// TIA Portal project "HeThongSanXuatTraXanh" (V16)

(* hardware
DEVICE "S7-1200 station_1"  S7-1200 Station
   slot 0: "Rack_0"  S7-1200 Rack  Rack  V1.0
   slot 1: "PLC_1"  CPU 1212C AC/DC/Rly  6ES7 212-1BE40-0XB0  V4.4
DEVICE "PC-System_1"  SIMATIC PC station
   slot 0: "SIMATIC PC station"  Rail  SIMATIC PC-Station  V1.0
      slot 125: "Stationmanager"  Station_Manager  V6.0.4
   slot 1: "HMI_RT_1"  WinCC RT Advanced  6AV2 104-0xxxx-xxxx  16.0.0.0
      slot 33792: "Computer interface"  Host interface
   slot 2: "IE general_1"  IE General  IE_CP  V8.2.0
*)

// ===== PLC "PLC_1"  CPU 1212C AC/DC/Rly =====

VAR_GLOBAL   // PLC tag table "Default tag table"
   "System_Byte" AT %MB1 : Byte;
   "FirstScan" AT %M1.0 : Bool;
   "DiagStatusUpdate" AT %M1.1 : Bool;
   "AlwaysTRUE" AT %M1.2 : Bool;
   "AlwaysFALSE" AT %M1.3 : Bool;
   "Clock_Byte" AT %MB0 : Byte;
   "Clock_10Hz" AT %M0.0 : Bool;
   "Clock_5Hz" AT %M0.1 : Bool;
   "Clock_2.5Hz" AT %M0.2 : Bool;
   "Clock_2Hz" AT %M0.3 : Bool;
   "Clock_1.25Hz" AT %M0.4 : Bool;
   "Clock_1Hz" AT %M0.5 : Bool;
   "Clock_0.625Hz" AT %M0.6 : Bool;
   "Clock_0.5Hz" AT %M0.7 : Bool;
   "alarm_word" AT %MW20 : Word;
   "alarm1" AT %M20.0 : Bool;
   "alarm2" AT %M20.1 : Bool;
END_VAR

VAR_GLOBAL   // PLC tag table "INPUT"
   "I_Mode" AT %I0.0 : Bool;
   "I_Auto_Run" AT %I0.1 : Bool;
   "I_Auto_Stop" AT %I0.2 : Bool;
   "I_BT1" AT %I0.3 : Bool;
   "I_BT2" AT %I0.4 : Bool;
   "I_BT3" AT %I0.5 : Bool;
   "I_BT4" AT %I0.6 : Bool;
   "I_BT5" AT %I0.7 : Bool;
   "I_BT6" AT %I1.0 : Bool;
   "I_Valve1" AT %I1.1 : Bool;
   "I_May_Hap" AT %I1.2 : Bool;
   "I_May_Vo" AT %I1.3 : Bool;
   "I_May_Say" AT %I1.4 : Bool;
   "I_May_Sang" AT %I1.5 : Bool;
   "I_May_Dong_Goi" AT %I1.6 : Bool;
   "IW_Loadcell" AT %IW64 : Int;
   "IW_Temp_Hap" AT %IW66 : Int;
   "IW_Temp_Say" AT %IW68 : Int;
END_VAR

VAR_GLOBAL   // PLC tag table "OUTPUT"
   "Q_Lamp_Auto" AT %Q0.0 : Bool;
   "Q_Lamp_Manu" AT %Q0.1 : Bool;
   "Q_Lamp_Auto_Running" AT %Q0.2 : Bool;
   "Q_BT1" AT %Q0.3 : Bool;
   "Q_BT2" AT %Q0.4 : Bool;
   "Q_BT3" AT %Q0.5 : Bool;
   "Q_BT4" AT %Q0.6 : Bool;
   "Q_BT5" AT %Q0.7 : Bool;
   "Q_BT6" AT %Q1.0 : Bool;
   "Q_Valve1" AT %Q1.1 : Bool;
   "Q_May_Hap" AT %Q1.2 : Bool;
   "Q_May_Vo" AT %Q1.3 : Bool;
   "Q_May_Say" AT %Q1.4 : Bool;
   "Q_May_Sang" AT %Q1.5 : Bool;
   "Q_May_Dong_Goi" AT %Q1.6 : Bool;
END_VAR

VAR_GLOBAL   // PLC tag table "MIEN_NHO"
   "Set_Weight" AT %MD100 : Real;
   "Set_Temp_Hap" AT %MD104 : Real;
   "Set_Temp_Say" AT %MD108 : Real;
   "Act_Weight" AT %MD200 : Real;
   "Act_Temp_Hap" AT %MD204 : Real;
   "Act_Temp_Say" AT %MD208 : Real;
   "Act_San_Luong" AT %MW212 : Int;
   "Simu_Temp" AT %MD220 : Real;
END_VAR

VAR_GLOBAL   // PLC tag table "TRUNG_GIAN"
   "Q_Auto_BT1" AT %M20.0 : Bool;
   "Q_Auto_BT2" AT %M20.1 : Bool;
   "Q_Auto_BT3" AT %M20.2 : Bool;
   "Q_Auto_BT4" AT %M20.3 : Bool;
   "Q_Auto_BT5" AT %M20.4 : Bool;
   "Q_Auto_BT6" AT %M20.5 : Bool;
   "Q_Auto_Valve1" AT %M20.6 : Bool;
   "Q_Auto_May_Hap" AT %M20.7 : Bool;
   "Q_Auto_May_Vo" AT %M21.0 : Bool;
   "Q_Auto_May_Say" AT %M21.1 : Bool;
   "Q_Auto_May_Sang" AT %M21.2 : Bool;
   "Q_Auto_May_Dong_Goi" AT %M21.3 : Bool;
   "Q_Manu_BT1" AT %M30.0 : Bool;
   "Q_Manu_BT2" AT %M30.1 : Bool;
   "Q_Manu_BT3" AT %M30.2 : Bool;
   "Q_Manu_BT4" AT %M30.3 : Bool;
   "Q_Manu_BT5" AT %M30.4 : Bool;
   "Q_Manu_BT6" AT %M30.5 : Bool;
   "Q_Manu_Valve1" AT %M30.6 : Bool;
   "Q_Manu_May_Hap" AT %M30.7 : Bool;
   "Q_Manu_May_Vo" AT %M31.0 : Bool;
   "Q_Manu_May_Say" AT %M31.1 : Bool;
   "Q_Manu_May_Sang" AT %M31.2 : Bool;
   "Q_Manu_May_Dong_Goi" AT %M31.3 : Bool;
END_VAR

VAR_GLOBAL   // PLC tag table "M"
   "M_Mode" AT %M10.0 : Bool;
   "M_Auto_Run" AT %M10.1 : Bool;
   "M_Auto_Stop" AT %M10.2 : Bool;
   "M_BT1" AT %M10.3 : Bool;
   "M_BT2" AT %M10.4 : Bool;
   "M_BT3" AT %M10.5 : Bool;
   "M_BT4" AT %M10.6 : Bool;
   "M_BT5" AT %M10.7 : Bool;
   "M_BT6" AT %M11.0 : Bool;
   "M_Valve1" AT %M11.1 : Bool;
   "M_May_Hap" AT %M11.2 : Bool;
   "M_May_Vo" AT %M11.3 : Bool;
   "M_May_Say" AT %M11.4 : Bool;
   "M_May_Sang" AT %M11.5 : Bool;
   "M_May_Dong_Goi" AT %M11.6 : Bool;
   "MW_Loadcell" AT %MW64 : Int;
   "MW_Temp_Hap" AT %MW66 : Int;
   "MW_Temp_Say" AT %MW68 : Int;
   "M_Simulation" AT %M5.0 : Bool;
END_VAR

VAR_GLOBAL   // PLC tag table "STEP"
   "STEP_1" AT %M40.0 : Bool;
   "STEP_2" AT %M40.1 : Bool;
   "STEP_3" AT %M40.2 : Bool;
   "STEP_4" AT %M40.3 : Bool;
   "STEP_5" AT %M40.4 : Bool;
   "STEP_6" AT %M40.5 : Bool;
   "STEP_7" AT %M40.6 : Bool;
   "STEP_8" AT %M40.7 : Bool;
   "STEP_9" AT %M41.0 : Bool;
   "STEP_10" AT %M41.1 : Bool;
   "STEP_11" AT %M41.2 : Bool;
END_VAR

VAR_GLOBAL   // PLC tag table "XUNG P"
   "P1" AT %M90.0 : Bool;
   "P2" AT %M90.1 : Bool;
   "P3" AT %M90.2 : Bool;
   "P4" AT %M90.3 : Bool;
   "P5" AT %M90.4 : Bool;
   "P6" AT %M90.5 : Bool;
   "P7" AT %M90.6 : Bool;
   "P8" AT %M90.7 : Bool;
   "P9" AT %M91.0 : Bool;
   "P10" AT %M91.1 : Bool;
   "P11" AT %M91.2 : Bool;
   "P12" AT %M91.3 : Bool;
   "P13" AT %M91.4 : Bool;
   "P14" AT %M91.5 : Bool;
   "P15" AT %M91.6 : Bool;
   "P16" AT %M91.7 : Bool;
   "P17" AT %M92.0 : Bool;
   "P18" AT %M92.1 : Bool;
   "P19" AT %M92.2 : Bool;
   "P20" AT %M92.3 : Bool;
END_VAR

// folder: System blocks/Program resources

DATA_BLOCK "TIMER_STEP2"   // DB1
{ S7_Optimized_Access := 'TRUE' }
AUTHOR : Simatic
FAMILY : IEC
NAME : IEC_TMR
VERSION : 1.0
// stored: InstanceOfName IEC_TIMER
"IEC_TIMER"
BEGIN
END_DATA_BLOCK

DATA_BLOCK "TIMER_STEP3"   // DB2
{ S7_Optimized_Access := 'TRUE' }
AUTHOR : Simatic
FAMILY : IEC
NAME : IEC_TMR
VERSION : 1.0
// stored: InstanceOfName IEC_TIMER
"IEC_TIMER"
BEGIN
END_DATA_BLOCK

DATA_BLOCK "TIMER_STEP4"   // DB3
{ S7_Optimized_Access := 'TRUE' }
AUTHOR : Simatic
FAMILY : IEC
NAME : IEC_TMR
VERSION : 1.0
// stored: InstanceOfName IEC_TIMER
"IEC_TIMER"
BEGIN
END_DATA_BLOCK

DATA_BLOCK "TIMER_STEP5"   // DB4
{ S7_Optimized_Access := 'TRUE' }
AUTHOR : Simatic
FAMILY : IEC
NAME : IEC_TMR
VERSION : 1.0
// stored: InstanceOfName IEC_TIMER
"IEC_TIMER"
BEGIN
END_DATA_BLOCK

DATA_BLOCK "TIMER_STEP6"   // DB5
{ S7_Optimized_Access := 'TRUE' }
AUTHOR : Simatic
FAMILY : IEC
NAME : IEC_TMR
VERSION : 1.0
// stored: InstanceOfName IEC_TIMER
"IEC_TIMER"
BEGIN
END_DATA_BLOCK

DATA_BLOCK "TIMER_STEP7"   // DB6
{ S7_Optimized_Access := 'TRUE' }
AUTHOR : Simatic
FAMILY : IEC
NAME : IEC_TMR
VERSION : 1.0
// stored: InstanceOfName IEC_TIMER
"IEC_TIMER"
BEGIN
END_DATA_BLOCK

DATA_BLOCK "TIMER_STEP8"   // DB7
{ S7_Optimized_Access := 'TRUE' }
AUTHOR : Simatic
FAMILY : IEC
NAME : IEC_TMR
VERSION : 1.0
// stored: InstanceOfName IEC_TIMER
"IEC_TIMER"
BEGIN
END_DATA_BLOCK

DATA_BLOCK "TIMER_STEP9"   // DB8
{ S7_Optimized_Access := 'TRUE' }
AUTHOR : Simatic
FAMILY : IEC
NAME : IEC_TMR
VERSION : 1.0
// stored: InstanceOfName IEC_TIMER
"IEC_TIMER"
BEGIN
END_DATA_BLOCK

DATA_BLOCK "TIMER_STEP10"   // DB9
{ S7_Optimized_Access := 'TRUE' }
AUTHOR : Simatic
FAMILY : IEC
NAME : IEC_TMR
VERSION : 1.0
// stored: InstanceOfName IEC_TIMER
"IEC_TIMER"
BEGIN
END_DATA_BLOCK

DATA_BLOCK "TIMER_STEP11"   // DB10
{ S7_Optimized_Access := 'TRUE' }
AUTHOR : Simatic
FAMILY : IEC
NAME : IEC_TMR
VERSION : 1.0
// stored: InstanceOfName IEC_TIMER
"IEC_TIMER"
BEGIN
END_DATA_BLOCK

// folder: (top level)

FUNCTION "FC_AUTO_MODE" : Void   // FC1, LAD
{ S7_Optimized_Access := 'TRUE' }
VERSION : 0.1
   VAR_TEMP   // added for the SCL form of the ladder/FBD networks
      _w1 : Bool;
      _w2 : Bool;
   END_VAR
BEGIN

REGION Network 1
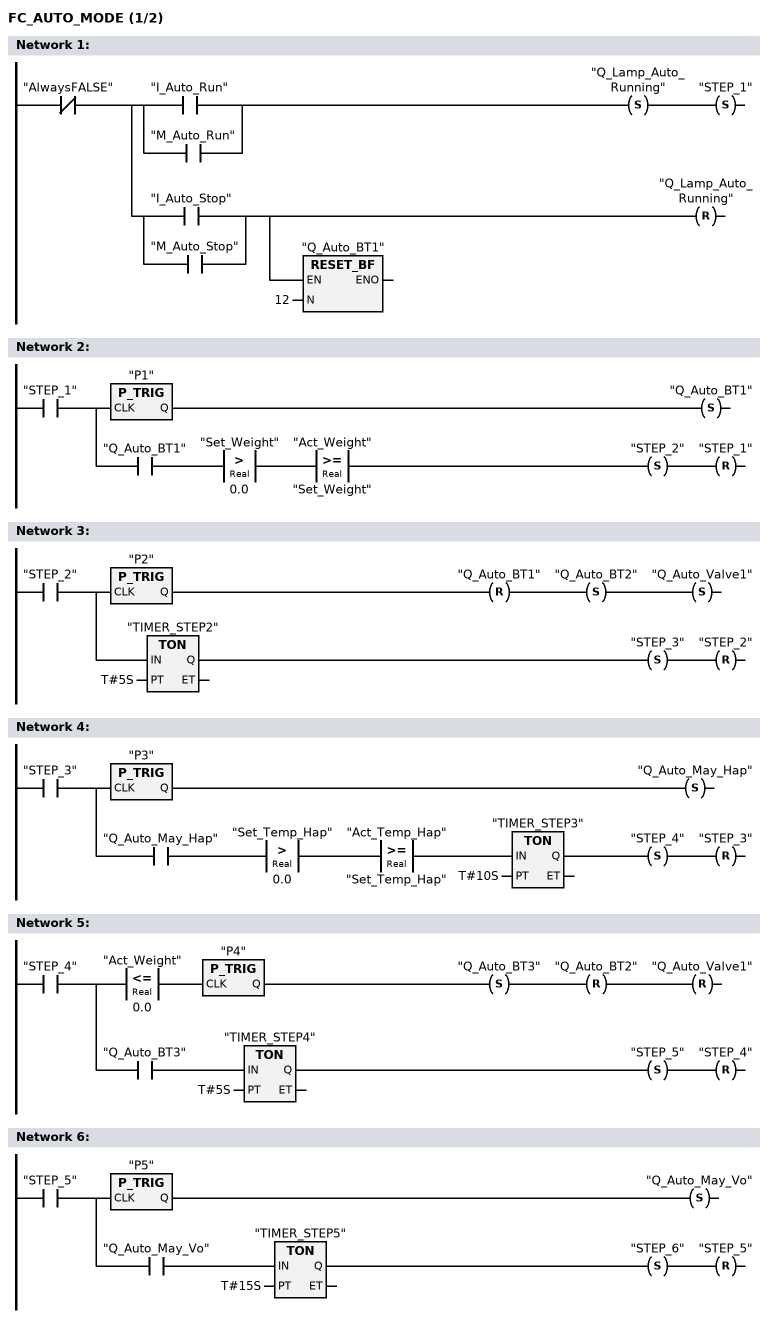
   // no SCL statement known for RBitfield: written as a call
   IF NOT "AlwaysFALSE" AND ("I_Auto_Run" OR "M_Auto_Run") THEN
       "Q_Lamp_Auto_Running" := TRUE;
       "STEP_1" := TRUE;
   END_IF;
   IF NOT "AlwaysFALSE" AND ("I_Auto_Stop" OR "M_Auto_Stop") THEN
       "Q_Lamp_Auto_Running" := FALSE;
       RESET_BF(operand := "Q_Auto_BT1", n := 12);
   END_IF;
END_REGION

REGION Network 2
   RUNG wire#powerrail
      Contact( "STEP_1" )
      wire#w1
      P_Trig( "P1" )
      S_Coil( "Q_Auto_BT1" )
   END_RUNG
   RUNG wire#w1
      Contact( "Q_Auto_BT1" )
      { S7_Templates := "SrcType := Real" } GT_Contact(in1 := "Set_Weight", in2 := 0.0)
      { S7_Templates := "SrcType := Real" } GE_Contact(in1 := "Act_Weight", in2 := "Set_Weight")
      S_Coil( "STEP_2" )
      R_Coil( "STEP_1" )
   END_RUNG
   // the same network as SCL:
   #_w1 := "STEP_1" AND NOT "P1";   // rising edge
   "P1" := "STEP_1";
   IF #_w1 THEN "Q_Auto_BT1" := TRUE; END_IF;
   IF "STEP_1" AND "Q_Auto_BT1" AND ("Set_Weight" > 0.0) AND ("Act_Weight" >= "Set_Weight") THEN
       "STEP_2" := TRUE;
       "STEP_1" := FALSE;
   END_IF;
END_REGION

REGION Network 3
   #_w1 := "STEP_2" AND NOT "P2";   // rising edge
   "P2" := "STEP_2";
   IF #_w1 THEN
       "Q_Auto_BT1" := FALSE;
       "Q_Auto_BT2" := TRUE;
       "Q_Auto_Valve1" := TRUE;
   END_IF;
   "TIMER_STEP2".TON(IN := "STEP_2", PT := T#5S);
   IF "TIMER_STEP2".Q THEN
       "STEP_3" := TRUE;
       "STEP_2" := FALSE;
   END_IF;
END_REGION

REGION Network 4
   #_w1 := "STEP_3" AND NOT "P3";   // rising edge
   "P3" := "STEP_3";
   IF #_w1 THEN "Q_Auto_May_Hap" := TRUE; END_IF;
   "TIMER_STEP3".TON(IN := "STEP_3" AND "Q_Auto_May_Hap" AND ("Set_Temp_Hap" > 0.0) AND ("Act_Temp_Hap" >= "Set_Temp_Hap"),
                     PT := T#10S);
   IF "TIMER_STEP3".Q THEN
       "STEP_4" := TRUE;
       "STEP_3" := FALSE;
   END_IF;
END_REGION

REGION Network 5
   #_w1 := "STEP_4" AND ("Act_Weight" <= 0.0);
   #_w2 := #_w1 AND NOT "P4";   // rising edge
   "P4" := #_w1;
   IF #_w2 THEN
       "Q_Auto_BT3" := TRUE;
       "Q_Auto_BT2" := FALSE;
       "Q_Auto_Valve1" := FALSE;
   END_IF;
   "TIMER_STEP4".TON(IN := "STEP_4" AND "Q_Auto_BT3", PT := T#5S);
   IF "TIMER_STEP4".Q THEN
       "STEP_5" := TRUE;
       "STEP_4" := FALSE;
   END_IF;
END_REGION

REGION Network 6
   #_w1 := "STEP_5" AND NOT "P5";   // rising edge
   "P5" := "STEP_5";
   IF #_w1 THEN "Q_Auto_May_Vo" := TRUE; END_IF;
   "TIMER_STEP5".TON(IN := "STEP_5" AND "Q_Auto_May_Vo", PT := T#15S);
   IF "TIMER_STEP5".Q THEN
       "STEP_6" := TRUE;
       "STEP_5" := FALSE;
   END_IF;
END_REGION

REGION Network 7
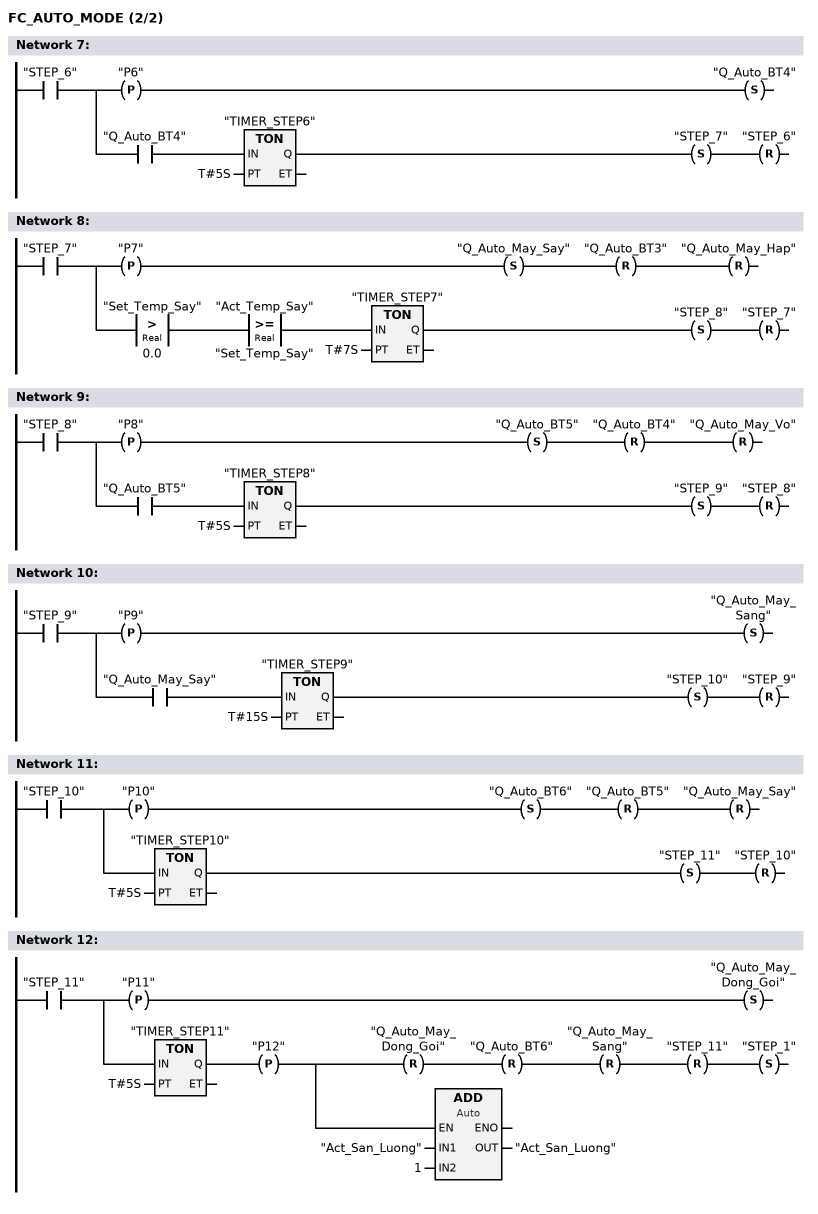
   #_w1 := "STEP_6" AND NOT "P6";   // rising edge
   "P6" := "STEP_6";
   IF #_w1 THEN "Q_Auto_BT4" := TRUE; END_IF;
   "TIMER_STEP6".TON(IN := "STEP_6" AND "Q_Auto_BT4", PT := T#5S);
   IF "TIMER_STEP6".Q THEN
       "STEP_7" := TRUE;
       "STEP_6" := FALSE;
   END_IF;
END_REGION

REGION Network 8
   #_w1 := "STEP_7" AND NOT "P7";   // rising edge
   "P7" := "STEP_7";
   IF #_w1 THEN
       "Q_Auto_May_Say" := TRUE;
       "Q_Auto_BT3" := FALSE;
       "Q_Auto_May_Hap" := FALSE;
   END_IF;
   "TIMER_STEP7".TON(IN := "STEP_7" AND ("Set_Temp_Say" > 0.0) AND ("Act_Temp_Say" >= "Set_Temp_Say"),
                     PT := T#7S);
   IF "TIMER_STEP7".Q THEN
       "STEP_8" := TRUE;
       "STEP_7" := FALSE;
   END_IF;
END_REGION

REGION Network 9
   #_w1 := "STEP_8" AND NOT "P8";   // rising edge
   "P8" := "STEP_8";
   IF #_w1 THEN
       "Q_Auto_BT5" := TRUE;
       "Q_Auto_BT4" := FALSE;
       "Q_Auto_May_Vo" := FALSE;
   END_IF;
   "TIMER_STEP8".TON(IN := "STEP_8" AND "Q_Auto_BT5", PT := T#5S);
   IF "TIMER_STEP8".Q THEN
       "STEP_9" := TRUE;
       "STEP_8" := FALSE;
   END_IF;
END_REGION

REGION Network 10
   #_w1 := "STEP_9" AND NOT "P9";   // rising edge
   "P9" := "STEP_9";
   IF #_w1 THEN "Q_Auto_May_Sang" := TRUE; END_IF;
   "TIMER_STEP9".TON(IN := "STEP_9" AND "Q_Auto_May_Say", PT := T#15S);
   IF "TIMER_STEP9".Q THEN
       "STEP_10" := TRUE;
       "STEP_9" := FALSE;
   END_IF;
END_REGION

REGION Network 11
   #_w1 := "STEP_10" AND NOT "P10";   // rising edge
   "P10" := "STEP_10";
   IF #_w1 THEN
       "Q_Auto_BT6" := TRUE;
       "Q_Auto_BT5" := FALSE;
       "Q_Auto_May_Say" := FALSE;
   END_IF;
   "TIMER_STEP10".TON(IN := "STEP_10", PT := T#5S);
   IF "TIMER_STEP10".Q THEN
       "STEP_11" := TRUE;
       "STEP_10" := FALSE;
   END_IF;
END_REGION

REGION Network 12
   #_w1 := "STEP_11" AND NOT "P11";   // rising edge
   "P11" := "STEP_11";
   IF #_w1 THEN "Q_Auto_May_Dong_Goi" := TRUE; END_IF;
   "TIMER_STEP11".TON(IN := "STEP_11", PT := T#5S);
   #_w2 := "TIMER_STEP11".Q AND NOT "P12";   // rising edge
   "P12" := "TIMER_STEP11".Q;
   IF #_w2 THEN
       "Q_Auto_May_Dong_Goi" := FALSE;
       "Q_Auto_BT6" := FALSE;
       "Q_Auto_May_Sang" := FALSE;
       "STEP_11" := FALSE;
       "STEP_1" := TRUE;
       "Act_San_Luong" := "Act_San_Luong" + 1;
   END_IF;
END_REGION
END_FUNCTION

FUNCTION "FC_MANUAL_MODE" : Void   // FC2, LAD
{ S7_Optimized_Access := 'TRUE' }
VERSION : 0.1
BEGIN

REGION Network 1
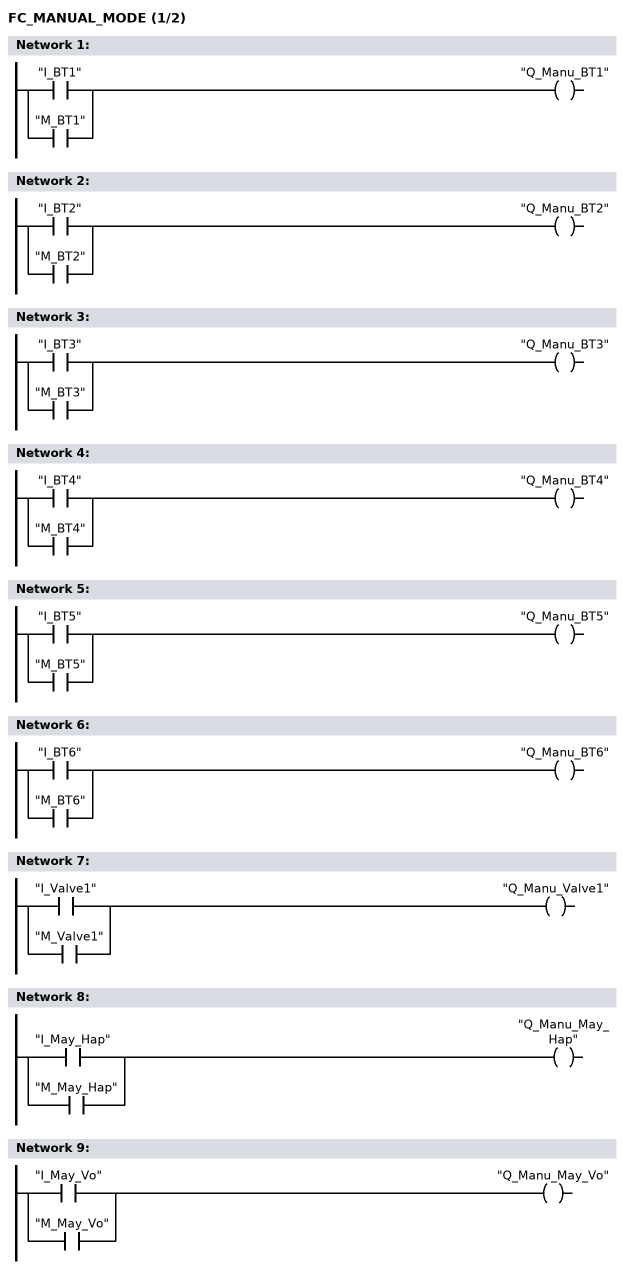
   RUNG wire#powerrail
      Contact( "I_BT1" )
      wire#w1
      Coil( "Q_Manu_BT1" )
   END_RUNG
   RUNG wire#powerrail
      Contact( "M_BT1" )
   END_RUNG wire#w1
   // the same network as SCL:
   "Q_Manu_BT1" := "I_BT1" OR "M_BT1";
END_REGION

REGION Network 2
   RUNG wire#powerrail
      Contact( "I_BT2" )
      wire#w1
      Coil( "Q_Manu_BT2" )
   END_RUNG
   RUNG wire#powerrail
      Contact( "M_BT2" )
   END_RUNG wire#w1
   // the same network as SCL:
   "Q_Manu_BT2" := "I_BT2" OR "M_BT2";
END_REGION

REGION Network 3
   RUNG wire#powerrail
      Contact( "I_BT3" )
      wire#w1
      Coil( "Q_Manu_BT3" )
   END_RUNG
   RUNG wire#powerrail
      Contact( "M_BT3" )
   END_RUNG wire#w1
   // the same network as SCL:
   "Q_Manu_BT3" := "I_BT3" OR "M_BT3";
END_REGION

REGION Network 4
   RUNG wire#powerrail
      Contact( "I_BT4" )
      wire#w1
      Coil( "Q_Manu_BT4" )
   END_RUNG
   RUNG wire#powerrail
      Contact( "M_BT4" )
   END_RUNG wire#w1
   // the same network as SCL:
   "Q_Manu_BT4" := "I_BT4" OR "M_BT4";
END_REGION

REGION Network 5
   RUNG wire#powerrail
      Contact( "I_BT5" )
      wire#w1
      Coil( "Q_Manu_BT5" )
   END_RUNG
   RUNG wire#powerrail
      Contact( "M_BT5" )
   END_RUNG wire#w1
   // the same network as SCL:
   "Q_Manu_BT5" := "I_BT5" OR "M_BT5";
END_REGION

REGION Network 6
   RUNG wire#powerrail
      Contact( "I_BT6" )
      wire#w1
      Coil( "Q_Manu_BT6" )
   END_RUNG
   RUNG wire#powerrail
      Contact( "M_BT6" )
   END_RUNG wire#w1
   // the same network as SCL:
   "Q_Manu_BT6" := "I_BT6" OR "M_BT6";
END_REGION

REGION Network 7
   RUNG wire#powerrail
      Contact( "I_Valve1" )
      wire#w1
      Coil( "Q_Manu_Valve1" )
   END_RUNG
   RUNG wire#powerrail
      Contact( "M_Valve1" )
   END_RUNG wire#w1
   // the same network as SCL:
   "Q_Manu_Valve1" := "I_Valve1" OR "M_Valve1";
END_REGION

REGION Network 8
   RUNG wire#powerrail
      Contact( "I_May_Hap" )
      wire#w1
      Coil( "Q_Manu_May_Hap" )
   END_RUNG
   RUNG wire#powerrail
      Contact( "M_May_Hap" )
   END_RUNG wire#w1
   // the same network as SCL:
   "Q_Manu_May_Hap" := "I_May_Hap" OR "M_May_Hap";
END_REGION

REGION Network 9
   RUNG wire#powerrail
      Contact( "I_May_Vo" )
      wire#w1
      Coil( "Q_Manu_May_Vo" )
   END_RUNG
   RUNG wire#powerrail
      Contact( "M_May_Vo" )
   END_RUNG wire#w1
   // the same network as SCL:
   "Q_Manu_May_Vo" := "I_May_Vo" OR "M_May_Vo";
END_REGION

REGION Network 10
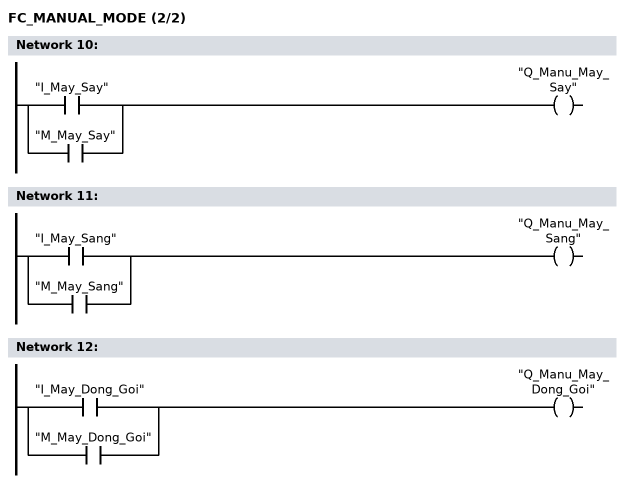
   RUNG wire#powerrail
      Contact( "I_May_Say" )
      wire#w1
      Coil( "Q_Manu_May_Say" )
   END_RUNG
   RUNG wire#powerrail
      Contact( "M_May_Say" )
   END_RUNG wire#w1
   // the same network as SCL:
   "Q_Manu_May_Say" := "I_May_Say" OR "M_May_Say";
END_REGION

REGION Network 11
   RUNG wire#powerrail
      Contact( "I_May_Sang" )
      wire#w1
      Coil( "Q_Manu_May_Sang" )
   END_RUNG
   RUNG wire#powerrail
      Contact( "M_May_Sang" )
   END_RUNG wire#w1
   // the same network as SCL:
   "Q_Manu_May_Sang" := "I_May_Sang" OR "M_May_Sang";
END_REGION

REGION Network 12
   RUNG wire#powerrail
      Contact( "I_May_Dong_Goi" )
      wire#w1
      Coil( "Q_Manu_May_Dong_Goi" )
   END_RUNG
   RUNG wire#powerrail
      Contact( "M_May_Dong_Goi" )
   END_RUNG wire#w1
   // the same network as SCL:
   "Q_Manu_May_Dong_Goi" := "I_May_Dong_Goi" OR "M_May_Dong_Goi";
END_REGION
END_FUNCTION

FUNCTION "FC_OUTPUT" : Void   // FC3, LAD
{ S7_Optimized_Access := 'TRUE' }
VERSION : 0.1
BEGIN

REGION Network 1
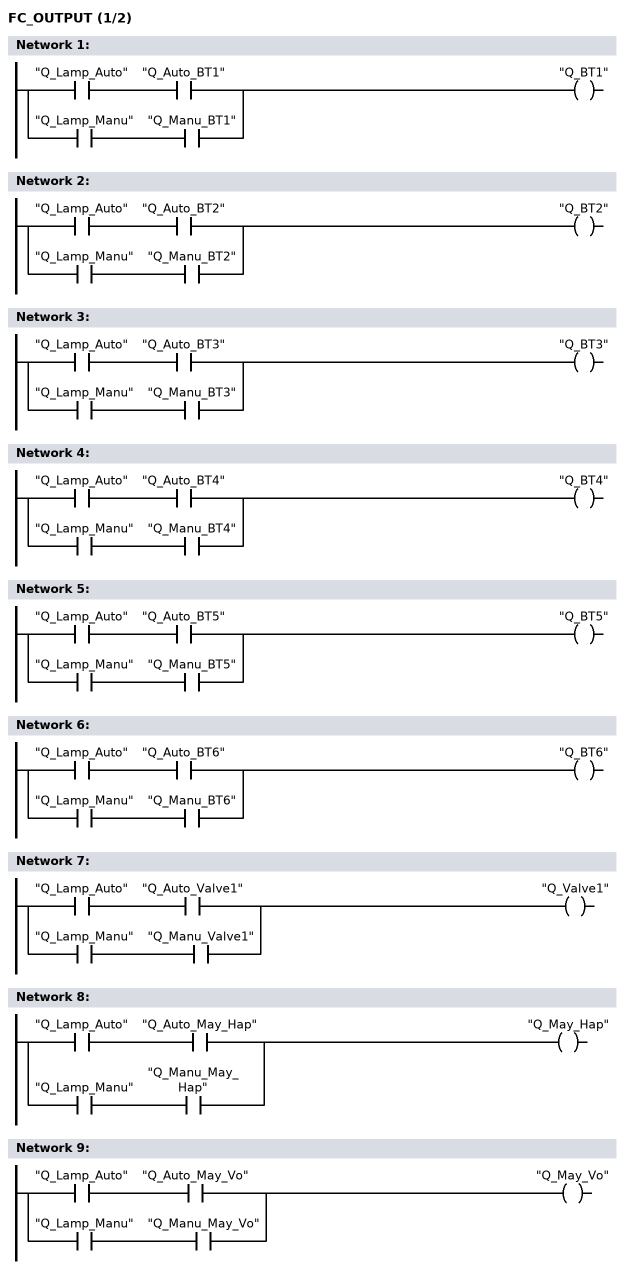
   RUNG wire#powerrail
      Contact( "Q_Lamp_Auto" )
      Contact( "Q_Auto_BT1" )
      wire#w1
      Coil( "Q_BT1" )
   END_RUNG
   RUNG wire#powerrail
      Contact( "Q_Lamp_Manu" )
      Contact( "Q_Manu_BT1" )
   END_RUNG wire#w1
   // the same network as SCL:
   "Q_BT1" := ("Q_Lamp_Auto" AND "Q_Auto_BT1") OR ("Q_Lamp_Manu" AND "Q_Manu_BT1");
END_REGION

REGION Network 2
   RUNG wire#powerrail
      Contact( "Q_Lamp_Auto" )
      Contact( "Q_Auto_BT2" )
      wire#w1
      Coil( "Q_BT2" )
   END_RUNG
   RUNG wire#powerrail
      Contact( "Q_Lamp_Manu" )
      Contact( "Q_Manu_BT2" )
   END_RUNG wire#w1
   // the same network as SCL:
   "Q_BT2" := ("Q_Lamp_Auto" AND "Q_Auto_BT2") OR ("Q_Lamp_Manu" AND "Q_Manu_BT2");
END_REGION

REGION Network 3
   RUNG wire#powerrail
      Contact( "Q_Lamp_Auto" )
      Contact( "Q_Auto_BT3" )
      wire#w1
      Coil( "Q_BT3" )
   END_RUNG
   RUNG wire#powerrail
      Contact( "Q_Lamp_Manu" )
      Contact( "Q_Manu_BT3" )
   END_RUNG wire#w1
   // the same network as SCL:
   "Q_BT3" := ("Q_Lamp_Auto" AND "Q_Auto_BT3") OR ("Q_Lamp_Manu" AND "Q_Manu_BT3");
END_REGION

REGION Network 4
   RUNG wire#powerrail
      Contact( "Q_Lamp_Auto" )
      Contact( "Q_Auto_BT4" )
      wire#w1
      Coil( "Q_BT4" )
   END_RUNG
   RUNG wire#powerrail
      Contact( "Q_Lamp_Manu" )
      Contact( "Q_Manu_BT4" )
   END_RUNG wire#w1
   // the same network as SCL:
   "Q_BT4" := ("Q_Lamp_Auto" AND "Q_Auto_BT4") OR ("Q_Lamp_Manu" AND "Q_Manu_BT4");
END_REGION

REGION Network 5
   RUNG wire#powerrail
      Contact( "Q_Lamp_Auto" )
      Contact( "Q_Auto_BT5" )
      wire#w1
      Coil( "Q_BT5" )
   END_RUNG
   RUNG wire#powerrail
      Contact( "Q_Lamp_Manu" )
      Contact( "Q_Manu_BT5" )
   END_RUNG wire#w1
   // the same network as SCL:
   "Q_BT5" := ("Q_Lamp_Auto" AND "Q_Auto_BT5") OR ("Q_Lamp_Manu" AND "Q_Manu_BT5");
END_REGION

REGION Network 6
   RUNG wire#powerrail
      Contact( "Q_Lamp_Auto" )
      Contact( "Q_Auto_BT6" )
      wire#w1
      Coil( "Q_BT6" )
   END_RUNG
   RUNG wire#powerrail
      Contact( "Q_Lamp_Manu" )
      Contact( "Q_Manu_BT6" )
   END_RUNG wire#w1
   // the same network as SCL:
   "Q_BT6" := ("Q_Lamp_Auto" AND "Q_Auto_BT6") OR ("Q_Lamp_Manu" AND "Q_Manu_BT6");
END_REGION

REGION Network 7
   RUNG wire#powerrail
      Contact( "Q_Lamp_Auto" )
      Contact( "Q_Auto_Valve1" )
      wire#w1
      Coil( "Q_Valve1" )
   END_RUNG
   RUNG wire#powerrail
      Contact( "Q_Lamp_Manu" )
      Contact( "Q_Manu_Valve1" )
   END_RUNG wire#w1
   // the same network as SCL:
   "Q_Valve1" := ("Q_Lamp_Auto" AND "Q_Auto_Valve1") OR ("Q_Lamp_Manu" AND "Q_Manu_Valve1");
END_REGION

REGION Network 8
   RUNG wire#powerrail
      Contact( "Q_Lamp_Auto" )
      Contact( "Q_Auto_May_Hap" )
      wire#w1
      Coil( "Q_May_Hap" )
   END_RUNG
   RUNG wire#powerrail
      Contact( "Q_Lamp_Manu" )
      Contact( "Q_Manu_May_Hap" )
   END_RUNG wire#w1
   // the same network as SCL:
   "Q_May_Hap" := ("Q_Lamp_Auto" AND "Q_Auto_May_Hap") OR ("Q_Lamp_Manu" AND "Q_Manu_May_Hap");
END_REGION

REGION Network 9
   RUNG wire#powerrail
      Contact( "Q_Lamp_Auto" )
      Contact( "Q_Auto_May_Vo" )
      wire#w1
      Coil( "Q_May_Vo" )
   END_RUNG
   RUNG wire#powerrail
      Contact( "Q_Lamp_Manu" )
      Contact( "Q_Manu_May_Vo" )
   END_RUNG wire#w1
   // the same network as SCL:
   "Q_May_Vo" := ("Q_Lamp_Auto" AND "Q_Auto_May_Vo") OR ("Q_Lamp_Manu" AND "Q_Manu_May_Vo");
END_REGION

REGION Network 10
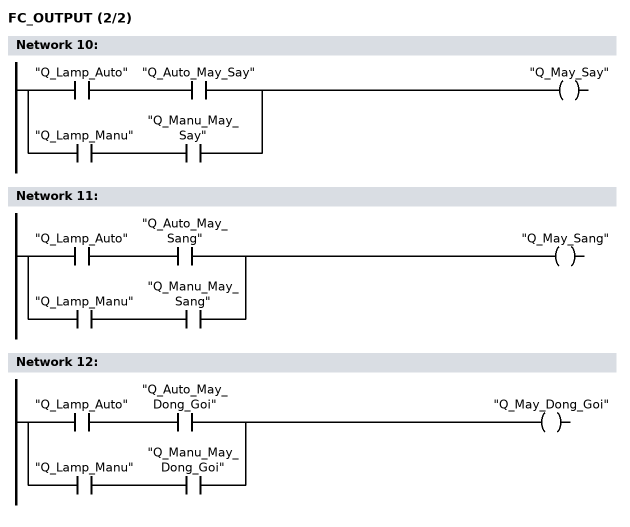
   RUNG wire#powerrail
      Contact( "Q_Lamp_Auto" )
      Contact( "Q_Auto_May_Say" )
      wire#w1
      Coil( "Q_May_Say" )
   END_RUNG
   RUNG wire#powerrail
      Contact( "Q_Lamp_Manu" )
      Contact( "Q_Manu_May_Say" )
   END_RUNG wire#w1
   // the same network as SCL:
   "Q_May_Say" := ("Q_Lamp_Auto" AND "Q_Auto_May_Say") OR ("Q_Lamp_Manu" AND "Q_Manu_May_Say");
END_REGION

REGION Network 11
   RUNG wire#powerrail
      Contact( "Q_Lamp_Auto" )
      Contact( "Q_Auto_May_Sang" )
      wire#w1
      Coil( "Q_May_Sang" )
   END_RUNG
   RUNG wire#powerrail
      Contact( "Q_Lamp_Manu" )
      Contact( "Q_Manu_May_Sang" )
   END_RUNG wire#w1
   // the same network as SCL:
   "Q_May_Sang" := ("Q_Lamp_Auto" AND "Q_Auto_May_Sang") OR ("Q_Lamp_Manu" AND "Q_Manu_May_Sang");
END_REGION

REGION Network 12
   RUNG wire#powerrail
      Contact( "Q_Lamp_Auto" )
      Contact( "Q_Auto_May_Dong_Goi" )
      wire#w1
      Coil( "Q_May_Dong_Goi" )
   END_RUNG
   RUNG wire#powerrail
      Contact( "Q_Lamp_Manu" )
      Contact( "Q_Manu_May_Dong_Goi" )
   END_RUNG wire#w1
   // the same network as SCL:
   "Q_May_Dong_Goi" := ("Q_Lamp_Auto" AND "Q_Auto_May_Dong_Goi") OR ("Q_Lamp_Manu" AND "Q_Manu_May_Dong_Goi");
END_REGION
END_FUNCTION

FUNCTION "FC_SIMULATION" : Void   // FC4, LAD
{ S7_Optimized_Access := 'TRUE' }
VERSION : 0.1
   VAR_TEMP   // added for the SCL form of the ladder/FBD networks
      _w1 : Bool;
      _w2 : Bool;
      _w3 : Bool;
      _w4 : Bool;
   END_VAR
BEGIN

REGION Network 1
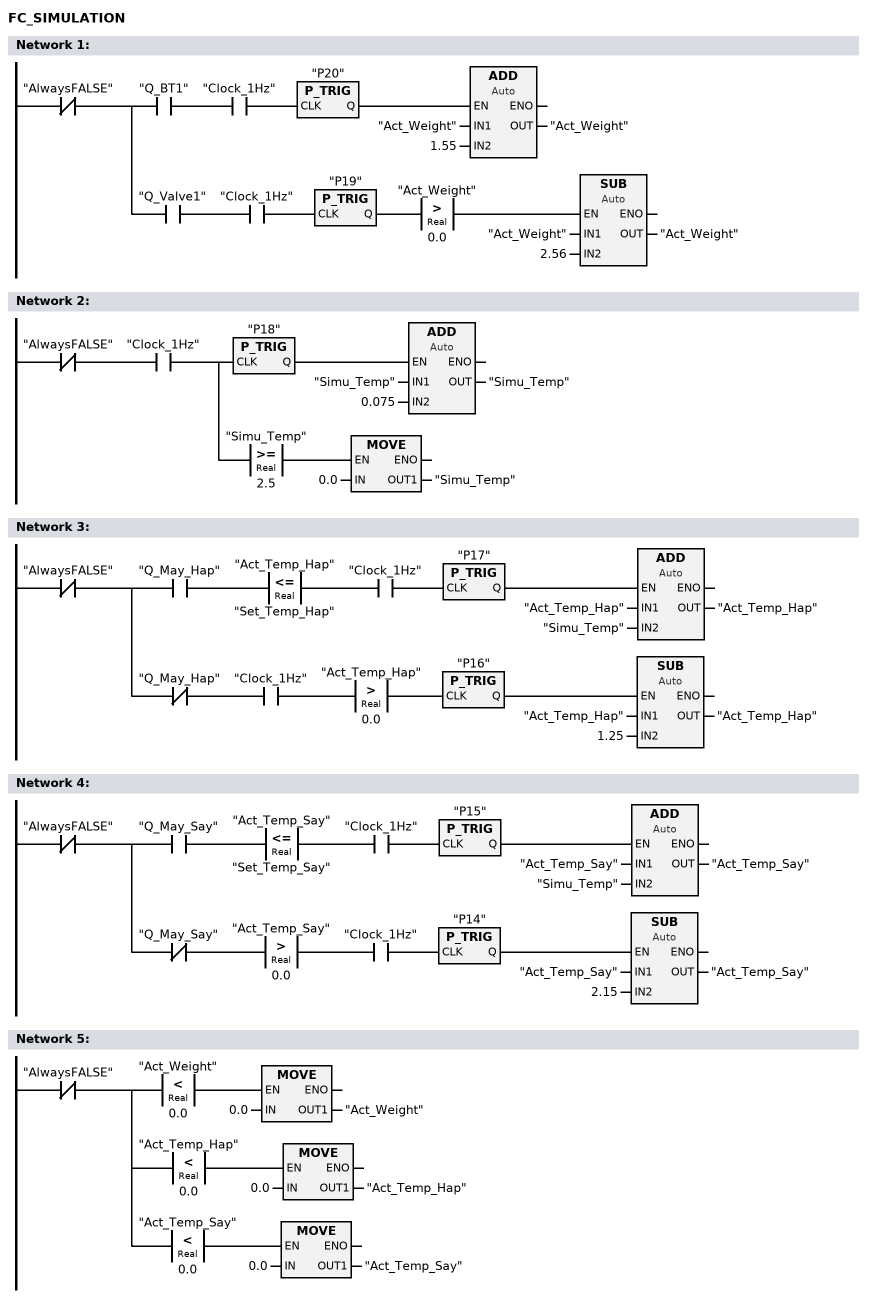
   RUNG wire#powerrail
      I_Contact( "AlwaysFALSE" )
      wire#w1
      Contact( "Q_BT1" )
      Contact( "Clock_1Hz" )
      P_Trig( "P20" )
      Add(in1 := "Act_Weight", in2 := 1.55, out => "Act_Weight")
   END_RUNG
   RUNG wire#w1
      Contact( "Q_Valve1" )
      Contact( "Clock_1Hz" )
      P_Trig( "P19" )
      { S7_Templates := "SrcType := Real" } GT_Contact(in1 := "Act_Weight", in2 := 0.0)
      Sub(in1 := "Act_Weight", in2 := 2.56, out => "Act_Weight")
   END_RUNG
   // the same network as SCL:
   #_w1 := NOT "AlwaysFALSE" AND "Q_BT1" AND "Clock_1Hz";
   #_w2 := #_w1 AND NOT "P20";   // rising edge
   "P20" := #_w1;
   IF #_w2 THEN "Act_Weight" := "Act_Weight" + 1.55; END_IF;
   #_w3 := NOT "AlwaysFALSE" AND "Q_Valve1" AND "Clock_1Hz";
   #_w4 := #_w3 AND NOT "P19";   // rising edge
   "P19" := #_w3;
   IF #_w4 AND ("Act_Weight" > 0.0) THEN "Act_Weight" := "Act_Weight" - 2.56; END_IF;
END_REGION

REGION Network 2
   RUNG wire#powerrail
      I_Contact( "AlwaysFALSE" )
      Contact( "Clock_1Hz" )
      wire#w1
      P_Trig( "P18" )
      Add(in1 := "Simu_Temp", in2 := 0.075, out => "Simu_Temp")
   END_RUNG
   RUNG wire#w1
      { S7_Templates := "SrcType := Real" } GE_Contact(in1 := "Simu_Temp", in2 := 2.5)
      Move(in := 0.0, out1 => "Simu_Temp")
   END_RUNG
   // the same network as SCL:
   #_w1 := NOT "AlwaysFALSE" AND "Clock_1Hz";
   #_w2 := #_w1 AND NOT "P18";   // rising edge
   "P18" := #_w1;
   IF #_w2 THEN "Simu_Temp" := "Simu_Temp" + 0.075; END_IF;
   IF #_w1 AND ("Simu_Temp" >= 2.5) THEN "Simu_Temp" := 0.0; END_IF;
END_REGION

REGION Network 3
   RUNG wire#powerrail
      I_Contact( "AlwaysFALSE" )
      wire#w1
      Contact( "Q_May_Hap" )
      { S7_Templates := "SrcType := Real" } LE_Contact(in1 := "Act_Temp_Hap", in2 := "Set_Temp_Hap")
      Contact( "Clock_1Hz" )
      P_Trig( "P17" )
      Add(in1 := "Act_Temp_Hap", in2 := "Simu_Temp", out => "Act_Temp_Hap")
   END_RUNG
   RUNG wire#w1
      I_Contact( "Q_May_Hap" )
      Contact( "Clock_1Hz" )
      { S7_Templates := "SrcType := Real" } GT_Contact(in1 := "Act_Temp_Hap", in2 := 0.0)
      P_Trig( "P16" )
      Sub(in1 := "Act_Temp_Hap", in2 := 1.25, out => "Act_Temp_Hap")
   END_RUNG
   // the same network as SCL:
   #_w1 := NOT "AlwaysFALSE" AND "Q_May_Hap" AND ("Act_Temp_Hap" <= "Set_Temp_Hap") AND "Clock_1Hz";
   #_w2 := #_w1 AND NOT "P17";   // rising edge
   "P17" := #_w1;
   IF #_w2 THEN "Act_Temp_Hap" := "Act_Temp_Hap" + "Simu_Temp"; END_IF;
   #_w3 := NOT "AlwaysFALSE" AND NOT "Q_May_Hap" AND "Clock_1Hz" AND ("Act_Temp_Hap" > 0.0);
   #_w4 := #_w3 AND NOT "P16";   // rising edge
   "P16" := #_w3;
   IF #_w4 THEN "Act_Temp_Hap" := "Act_Temp_Hap" - 1.25; END_IF;
END_REGION

REGION Network 4
   RUNG wire#powerrail
      I_Contact( "AlwaysFALSE" )
      wire#w1
      Contact( "Q_May_Say" )
      { S7_Templates := "SrcType := Real" } LE_Contact(in1 := "Act_Temp_Say", in2 := "Set_Temp_Say")
      Contact( "Clock_1Hz" )
      P_Trig( "P15" )
      Add(in1 := "Act_Temp_Say", in2 := "Simu_Temp", out => "Act_Temp_Say")
   END_RUNG
   RUNG wire#w1
      I_Contact( "Q_May_Say" )
      { S7_Templates := "SrcType := Real" } GT_Contact(in1 := "Act_Temp_Say", in2 := 0.0)
      Contact( "Clock_1Hz" )
      P_Trig( "P14" )
      Sub(in1 := "Act_Temp_Say", in2 := 2.15, out => "Act_Temp_Say")
   END_RUNG
   // the same network as SCL:
   #_w1 := NOT "AlwaysFALSE" AND "Q_May_Say" AND ("Act_Temp_Say" <= "Set_Temp_Say") AND "Clock_1Hz";
   #_w2 := #_w1 AND NOT "P15";   // rising edge
   "P15" := #_w1;
   IF #_w2 THEN "Act_Temp_Say" := "Act_Temp_Say" + "Simu_Temp"; END_IF;
   #_w3 := NOT "AlwaysFALSE" AND NOT "Q_May_Say" AND ("Act_Temp_Say" > 0.0) AND "Clock_1Hz";
   #_w4 := #_w3 AND NOT "P14";   // rising edge
   "P14" := #_w3;
   IF #_w4 THEN "Act_Temp_Say" := "Act_Temp_Say" - 2.15; END_IF;
END_REGION

REGION Network 5
   RUNG wire#powerrail
      I_Contact( "AlwaysFALSE" )
      wire#w1
      { S7_Templates := "SrcType := Real" } LT_Contact(in1 := "Act_Weight", in2 := 0.0)
      Move(in := 0.0, out1 => "Act_Weight")
   END_RUNG
   RUNG wire#w1
      { S7_Templates := "SrcType := Real" } LT_Contact(in1 := "Act_Temp_Hap", in2 := 0.0)
      Move(in := 0.0, out1 => "Act_Temp_Hap")
   END_RUNG
   RUNG wire#w1
      { S7_Templates := "SrcType := Real" } LT_Contact(in1 := "Act_Temp_Say", in2 := 0.0)
      Move(in := 0.0, out1 => "Act_Temp_Say")
   END_RUNG
   // the same network as SCL:
   IF NOT "AlwaysFALSE" AND ("Act_Weight" < 0.0) THEN "Act_Weight" := 0.0; END_IF;
   IF NOT "AlwaysFALSE" AND ("Act_Temp_Hap" < 0.0) THEN "Act_Temp_Hap" := 0.0; END_IF;
   IF NOT "AlwaysFALSE" AND ("Act_Temp_Say" < 0.0) THEN "Act_Temp_Say" := 0.0; END_IF;
END_REGION
END_FUNCTION

FUNCTION "FC_READ_ANALOG" : Void   // FC5, LAD
{ S7_Optimized_Access := 'TRUE' }
VERSION : 0.1
   VAR_TEMP
      Analog_1 : Real;
      Analog_2 : Real;
      Analog_3 : Real;
   END_VAR
BEGIN

REGION Network 1
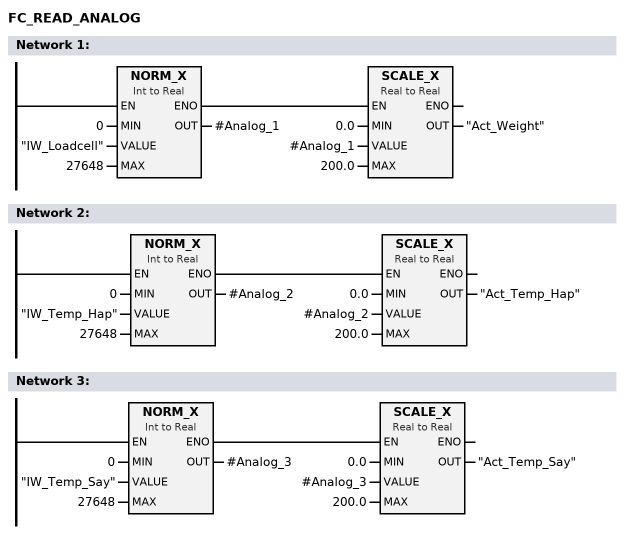
   RUNG wire#powerrail
      { S7_Templates := "[SrcType := Int, DestType := Real]" } Normalize(min := 0, value := "IW_Loadcell", max := 27648, out => #Analog_1)
      { S7_Templates := "[SrcType := Real, DestType := Real]" } Scale(min := 0.0, value := #Analog_1, max := 200.0, out => "Act_Weight")
   END_RUNG
   // the same network as SCL:
   #Analog_1 := NORM_X(MIN := 0, VALUE := "IW_Loadcell", MAX := 27648);
   "Act_Weight" := SCALE_X(MIN := 0.0, VALUE := #Analog_1, MAX := 200.0);
END_REGION

REGION Network 2
   RUNG wire#powerrail
      { S7_Templates := "[SrcType := Int, DestType := Real]" } Normalize(min := 0, value := "IW_Temp_Hap", max := 27648, out => #Analog_2)
      { S7_Templates := "[SrcType := Real, DestType := Real]" } Scale(min := 0.0, value := #Analog_2, max := 200.0, out => "Act_Temp_Hap")
   END_RUNG
   // the same network as SCL:
   #Analog_2 := NORM_X(MIN := 0, VALUE := "IW_Temp_Hap", MAX := 27648);
   "Act_Temp_Hap" := SCALE_X(MIN := 0.0, VALUE := #Analog_2, MAX := 200.0);
END_REGION

REGION Network 3
   RUNG wire#powerrail
      { S7_Templates := "[SrcType := Int, DestType := Real]" } Normalize(min := 0, value := "IW_Temp_Say", max := 27648, out => #Analog_3)
      { S7_Templates := "[SrcType := Real, DestType := Real]" } Scale(min := 0.0, value := #Analog_3, max := 200.0, out => "Act_Temp_Say")
   END_RUNG
   // the same network as SCL:
   #Analog_3 := NORM_X(MIN := 0, VALUE := "IW_Temp_Say", MAX := 27648);
   "Act_Temp_Say" := SCALE_X(MIN := 0.0, VALUE := #Analog_3, MAX := 200.0);
END_REGION
END_FUNCTION

ORGANIZATION_BLOCK "Main"   // OB1, LAD, ProgramCycle
TITLE = "Main Program Sweep (Cycle)"
{ S7_Optimized_Access := 'TRUE' }
VERSION : 0.1
   VAR_INPUT
      Initial_Call : Bool;   // Initial call of this OB
      Remanence : Bool;   // =True, if remanent data are available
   END_VAR
BEGIN

REGION Network 1: Chế độ vận hành
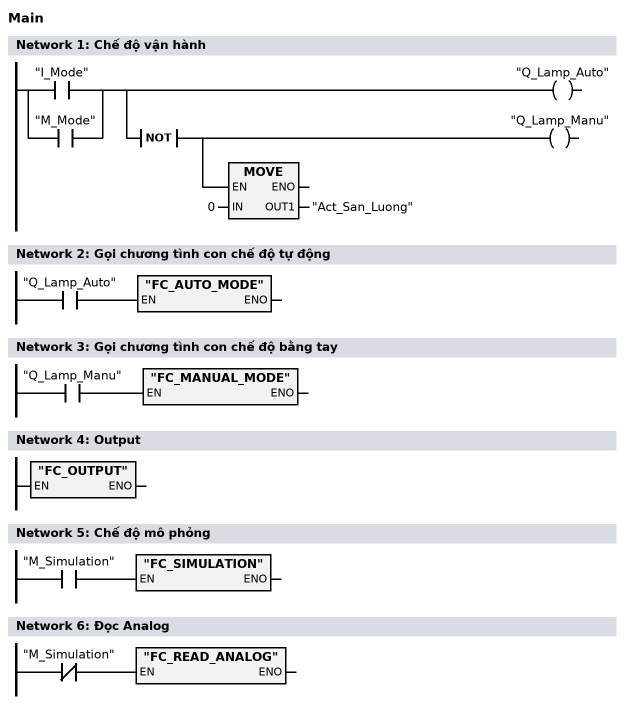
   RUNG wire#powerrail
      Contact( "I_Mode" )
      wire#w1
      Coil( "Q_Lamp_Auto" )
   END_RUNG
   RUNG wire#powerrail
      Contact( "M_Mode" )
   END_RUNG wire#w1
   RUNG wire#w1
      Not()
      wire#w2
      Coil( "Q_Lamp_Manu" )
   END_RUNG
   RUNG wire#w2
      Move(in := 0, out1 => "Act_San_Luong")
   END_RUNG
   // the same network as SCL:
   "Q_Lamp_Auto" := "I_Mode" OR "M_Mode";
   "Q_Lamp_Manu" := NOT "Q_Lamp_Auto";
   IF NOT "Q_Lamp_Auto" THEN "Act_San_Luong" := 0; END_IF;
END_REGION

REGION Network 2: Gọi chương tình con chế độ tự động
   RUNG wire#powerrail
      Contact( "Q_Lamp_Auto" )
      "FC_AUTO_MODE"()
   END_RUNG
   // the same network as SCL:
   IF "Q_Lamp_Auto" THEN "FC_AUTO_MODE"(); END_IF;
END_REGION

REGION Network 3: Gọi chương tình con chế độ bằng tay
   RUNG wire#powerrail
      Contact( "Q_Lamp_Manu" )
      "FC_MANUAL_MODE"()
   END_RUNG
   // the same network as SCL:
   IF "Q_Lamp_Manu" THEN "FC_MANUAL_MODE"(); END_IF;
END_REGION

REGION Network 4: Output
   RUNG wire#powerrail
      "FC_OUTPUT"()
   END_RUNG
   // the same network as SCL:
   "FC_OUTPUT"();
END_REGION

REGION Network 5: Chế độ mô phỏng
   RUNG wire#powerrail
      Contact( "M_Simulation" )
      "FC_SIMULATION"()
   END_RUNG
   // the same network as SCL:
   IF "M_Simulation" THEN "FC_SIMULATION"(); END_IF;
END_REGION

REGION Network 6: Đọc Analog
   RUNG wire#powerrail
      I_Contact( "M_Simulation" )
      "FC_READ_ANALOG"()
   END_RUNG
   // the same network as SCL:
   IF NOT "M_Simulation" THEN "FC_READ_ANALOG"(); END_IF;
END_REGION
END_ORGANIZATION_BLOCK

ORGANIZATION_BLOCK "Startup"   // OB100, LAD, Startup
TITLE = "Complete Restart"
{ S7_Optimized_Access := 'TRUE' }
VERSION : 0.1
   VAR_INPUT
      LostRetentive : Bool;   // True if retentive data are lost
      LostRTC : Bool;   // True if date and time are lost
   END_VAR
BEGIN

REGION Network 1
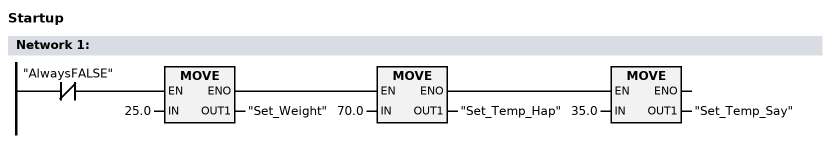
   RUNG wire#powerrail
      I_Contact( "AlwaysFALSE" )
      Move(in := 25.0, out1 => "Set_Weight")
      Move(in := 70.0, out1 => "Set_Temp_Hap")
      Move(in := 35.0, out1 => "Set_Temp_Say")
   END_RUNG
   // the same network as SCL:
   IF NOT "AlwaysFALSE" THEN
       "Set_Weight" := 25.0;
       "Set_Temp_Hap" := 70.0;
       "Set_Temp_Say" := 35.0;
   END_IF;
END_REGION
END_ORGANIZATION_BLOCK

(* ===== HMI "HMI_RT_1" =====
system functions are stored by id; their names below are inferred from use
connection "HMI_Connection_1": ETHERNET, S7_1200_OMS

HMI tags "Default tag table"
   "M_Mode" : Bool = PLC M_Mode AT %M10.0, 1 s
   "M_Simulation" : Bool = PLC M_Simulation AT %M5.0, 1 s
   "M_Auto_Run" : Bool = PLC M_Auto_Run AT %M10.1, 1 s
   "Q_Lamp_Auto_Running" : Bool = PLC Q_Lamp_Auto_Running AT %Q0.2, 1 s
   "Set_Weight" : Real = PLC Set_Weight AT %MD100, 1 s
   "Set_Temp_Say" : Real = PLC Set_Temp_Say AT %MD108, 1 s
   "Set_Temp_Hap" : Real = PLC Set_Temp_Hap AT %MD104, 1 s
   "Act_San_Luong" : Int = PLC Act_San_Luong AT %MW212, 1 s
   "Act_Temp_Say" : Real = PLC Act_Temp_Say AT %MD208, 1 s
   "Act_Temp_Hap" : Real = PLC Act_Temp_Hap AT %MD204, 1 s
   "Act_Weight" : Real = PLC Act_Weight AT %MD200, 1 s
   "M_BT1" : Bool = PLC M_BT1 AT %M10.3, 1 s
   "M_Valve1" : Bool = PLC M_Valve1 AT %M11.1, 1 s
   "M_BT2" : Bool = PLC M_BT2 AT %M10.4, 1 s
   "M_May_Hap" : Bool = PLC M_May_Hap AT %M11.2, 1 s
   "M_BT3" : Bool = PLC M_BT3 AT %M10.5, 1 s
   "M_BT4" : Bool = PLC M_BT4 AT %M10.6, 1 s
   "M_BT5" : Bool = PLC M_BT5 AT %M10.7, 1 s
   "M_May_Vo" : Bool = PLC M_May_Vo AT %M11.3, 1 s
   "M_May_Say" : Bool = PLC M_May_Say AT %M11.4, 1 s
   "M_May_Sang" : Bool = PLC M_May_Sang AT %M11.5, 1 s
   "M_BT6" : Bool = PLC M_BT6 AT %M11.0, 1 s
   "M_May_Dong_Goi" : Bool = PLC M_May_Dong_Goi AT %M11.6, 1 s
   "Q_Lamp_Manu" : Bool = PLC Q_Lamp_Manu AT %Q0.1, 1 s
   "Q_Lamp_Auto" : Bool = PLC Q_Lamp_Auto AT %Q0.0, 1 s
   "Q_BT1" : Bool = PLC Q_BT1 AT %Q0.3, 1 s
   "Q_Valve1" : Bool = PLC Q_Valve1 AT %Q1.1, 1 s
   "Q_BT2" : Bool = PLC Q_BT2 AT %Q0.4, 1 s
   "Q_May_Hap" : Bool = PLC Q_May_Hap AT %Q1.2, 1 s
   "Q_BT3" : Bool = PLC Q_BT3 AT %Q0.5, 1 s
   "Q_May_Vo" : Bool = PLC Q_May_Vo AT %Q1.3, 1 s
   "Q_BT4" : Bool = PLC Q_BT4 AT %Q0.6, 1 s
   "Q_May_Say" : Bool = PLC Q_May_Say AT %Q1.4, 1 s
   "Q_BT5" : Bool = PLC Q_BT5 AT %Q0.7, 1 s
   "Q_May_Sang" : Bool = PLC Q_May_Sang AT %Q1.5, 1 s
   "Q_BT6" : Bool = PLC Q_BT6 AT %Q1.0, 1 s
   "Q_May_Dong_Goi" : Bool = PLC Q_May_Dong_Goi AT %Q1.6, 1 s
   "M_Auto_Stop" : Bool = PLC M_Auto_Stop AT %M10.2, 1 s
   "alarm_word" : Word = PLC alarm_word AT %MW20, 1 s
   "alarm1" : Bool = PLC alarm1 AT %M20.0, 1 s
   "alarm2" : Bool = PLC alarm2 AT %M20.1, 1 s

discrete alarms
   1: 'overheat', class Warnings, trigger "alarm_word" bit 8
   2: 'broken_equipment', class Warnings, trigger "alarm_word" bit 9

screen "Screen_1" 1440x900
   TextField "Text field_2" at 51,219 size 116x40; Text 'Băng tải 1'
   SymbolLibrary "Symbol library_3" at 190,155 size 89x140
   SymbolLibrary "Symbol library_4" at 216,292 size 70x65
      Appearance <- "Q_Valve1"
   TextField "Text field_3" at 285,205 size 107x40; Text 'Bồn cân'
   TextField "Text field_4" at 158,320 size 71x40; Text 'Van 1'
   SymbolLibrary "Symbol library_5" at 185,374 size 186x53
      Appearance <- "Q_BT2"
   SymbolLibrary "Symbol library_6" at 191,433 size 89x67
      Appearance <- "Q_BT2"
   TextField "Text field_5" at 194,502 size 124x40; Text 'Băng tải 2'
   SymbolLibrary "Symbol library_7" at 348,430 size 157x96
      Appearance <- "Q_May_Hap"
   TextField "Text field_6" at 376,531 size 115x40; Text 'Máy hấp'
   SymbolLibrary "Symbol library_8" at 492,335 size 199x181
      Appearance <- "Q_BT3"
   SymbolLibrary "Symbol library_9" at 675,323 size 127x117
      Appearance <- "Q_May_Vo"
   TextField "Text field_7" at 707,292 size 118x40; Text 'Mày vò'
   TextField "Text field_8" at 559,530 size 128x40; Text 'Băng tải 3'
   SymbolLibrary "Symbol library_10" at 735,454 size 186x53
      Appearance <- "Q_BT4"
   SymbolLibrary "Symbol library_11" at 740,513 size 89x67
      Appearance <- "Q_BT4"
   TextField "Text field_9" at 743,582 size 140x40; Text 'Băng tải 4'
   SymbolLibrary "Symbol library_12" at 884,429 size 104x95
      Appearance <- "Q_May_Say"
   TextField "Text field_10" at 913,399 size 134x40; Text 'Máy sấy'
   SymbolLibrary "Symbol library_13" at 956,490 size 186x53
      Appearance <- "Q_BT5"
   SymbolLibrary "Symbol library_14" at 961,550 size 89x67
      Appearance <- "Q_BT5"
   TextField "Text field_11" at 964,619 size 144x40; Text 'Băng tải 5'
   SymbolLibrary "Symbol library_15" at 1096,547 size 89x109
      Appearance <- "Q_May_Sang"
   TextField "Text field_12" at 1188,593 size 155x40; Text 'Máy sàng'
   SymbolLibrary "Symbol library_16" at 1143,675 size 186x53
      Appearance <- "Q_BT6"
   SymbolLibrary "Symbol library_17" at 1149,734 size 89x67
      Appearance <- "Q_BT6"
   TextField "Text field_13" at 1153,812 size 136x40; Text 'Băng tải 6'
   SymbolLibrary "Symbol library_18" at 1290,713 size 111x154
      Appearance <- "Q_May_Dong_Goi"
   TextField "Text field_14" at 1281,635 size 159x40; Text 'Máy đóng gói'
   TextField "Text field_1" at 452,21 size 721x76; Text 'Hệ thống sản xuất trà xanh'
   IOField "I/O field_1" at 285,245 size 96x32; Authorization "onlyread"; FormatPattern 999999999.999
      ProcessValue <- "Act_Weight"
   TextField "Text field_15" at 385,249 size 87x40; Text 'kg'
   IOField "I/O field_2" at 348,563 size 96x32; Authorization "onlyread"; FormatPattern 999999999.999
      ProcessValue <- "Act_Temp_Hap"
   TextField "Text field_16" at 448,567 size 99x40; Text 'độ'
   IOField "I/O field_3" at 883,357 size 96x32; Authorization "onlyread"; FormatPattern 999999999.999
      ProcessValue <- "Act_Temp_Say"
   TextField "Text field_17" at 983,361 size 79x40; Text 'độ'
   SymbolLibrary "Symbol library_19" at 42,88 size 186x53
      Appearance <- "Q_BT1"
   SymbolLibrary "Symbol library_1" at 51,148 size 89x67
      Appearance <- "Q_BT1"
   Switch "Switch_1" at 1130,160 size 211x88; CaptionText 'mô phỏng'; TextOff 'OFF'; TextOn 'ON'; Authorization "giamdoc"
      ProcessValue <- "M_Simulation"
      on SwitchOff: ResetBit("M_Simulation")
      on SwitchOn: SetBit("M_Simulation")
   Switch "Switch_2" at 1130,58 size 211x88; TextOn 'tự động'; CaptionText 'Chế độ vận hành'; TextOff 'bằng tay'; Authorization "giamdoc"
      on SwitchOn: SetBit("M_Mode")
      on SwitchOff: ResetBit("M_Mode")
      ProcessValue <- "M_Mode"
   Button "Button_1" at 1127,291 size 96x32; TextOff 'Start'; Authorization "giamdoc"
      on Press: SetBit("M_Auto_Run")
      on Release: ResetBit("M_Auto_Run")
      Appearance <- "Q_Lamp_Auto_Running"
   Button "Button_2" at 1245,291 size 96x32; TextOff 'Stop'; Authorization "giamdoc"
      on Press: SetBit("M_Auto_Stop")
      on Release: ResetBit("M_Auto_Stop")
      Appearance <- "Q_Lamp_Auto_Running"
   IOField "I/O field_4" at 773,81 size 160x32; Authorization "giamdoc"; FormatPattern 999999999.999; Unit kg
      ProcessValue <- "Set_Weight"
   IOField "I/O field_5" at 773,137 size 161x32; Authorization "giamdoc"; FormatPattern 999999999.999; Unit độ
      ProcessValue <- "Set_Temp_Hap"
   IOField "I/O field_6" at 773,196 size 162x32; Authorization "giamdoc"; FormatPattern 999999999.999; Unit độ
      ProcessValue <- "Set_Temp_Say"
   TextField "Text field_18" at 644,81 size 134x40; Text 'Trọng lượng'
   TextField "Text field_19" at 646,137 size 95x40; Text 'ND hấp'
   TextField "Text field_20" at 643,196 size 98x40; Text 'ND sấy'
   IOField "I/O field_7" at 714,672 size 96x32; Authorization "onlyread"; FormatPattern 99999
      ProcessValue <- "Act_San_Luong"
   TextField "Text field_21" at 811,673 size 45x40; Text 'SP'
   Switch "Switch_3" at 46,245 size 89x40; CaptionText 'Switch'; TextOff 'OFF'; TextOn 'ON'; Authorization "khau1"
      on SwitchOn: SetBit("M_BT1")
      on SwitchOff: ResetBit("M_BT1")
      ProcessValue <- "M_BT1"
   Switch "Switch_5" at 190,526 size 89x40; TextOn 'ON'; CaptionText 'Switch'; TextOff 'OFF'; Authorization "khau2"
      on SwitchOff: ResetBit("M_BT2")
      on SwitchOn: SetBit("M_BT2")
      ProcessValue <- "M_BT2"
   Switch "Switch_6" at 423,386 size 89x40; TextOn 'ON'; CaptionText 'Switch'; TextOff 'OFF'; Authorization "khau2"
      on SwitchOn: SetBit("M_May_Hap")
      on SwitchOff: ResetBit("M_May_Hap")
      ProcessValue <- "M_May_Hap"
   Switch "Switch_7" at 552,558 size 89x40; TextOn 'ON'; CaptionText 'Switch'; TextOff 'OFF'; Authorization "khau3"
      on SwitchOn: SetBit("M_BT3")
      on SwitchOff: ResetBit("M_BT3")
      ProcessValue <- "M_BT3"
   Switch "Switch_8" at 847,548 size 89x40; TextOn 'ON'; CaptionText 'Switch'; TextOff 'OFF'; Authorization "khau4"
      on SwitchOff: ResetBit("M_BT4")
      on SwitchOn: SetBit("M_BT4")
      ProcessValue <- "M_BT4"
   Switch "Switch_9" at 956,646 size 89x40; TextOn 'ON'; CaptionText 'Switch'; TextOff 'OFF'; Authorization "khau5"
      on SwitchOn: SetBit("M_BT5")
      on SwitchOff: ResetBit("M_BT5")
      ProcessValue <- "M_BT5"
   Switch "Switch_10" at 601,291 size 89x40; TextOn 'ON'; CaptionText 'Switch'; TextOff 'OFF'; Authorization "khau3"
      on SwitchOff: ResetBit("M_May_Vo")
      on SwitchOn: SetBit("M_May_Vo")
      ProcessValue <- "M_May_Vo"
   Switch "Switch_11" at 998,414 size 89x40; TextOn 'ON'; CaptionText 'Switch'; TextOff 'OFF'; Authorization "khau4"
      on SwitchOn: SetBit("M_May_Say")
      on SwitchOff: ResetBit("M_May_Say")
      ProcessValue <- "M_May_Say"
   Switch "Switch_12" at 1201,516 size 89x40; TextOn 'ON'; CaptionText 'Switch'; TextOff 'OFF'; Authorization "khau5"
      on SwitchOff: ResetBit("M_May_Sang")
      on SwitchOn: SetBit("M_May_Sang")
      ProcessValue <- "M_May_Sang"
   Switch "Switch_13" at 1034,735 size 89x40; TextOn 'ON'; CaptionText 'Switch'; TextOff 'OFF'; Authorization "khau6"
      on SwitchOff: ResetBit("M_BT6")
      on SwitchOn: SetBit("M_BT6")
      ProcessValue <- "M_BT6"
   Switch "Switch_14" at 1333,658 size 89x40; TextOn 'ON'; CaptionText 'Switch'; TextOff 'OFF'; Authorization "khau6"
      on SwitchOn: SetBit("M_May_Dong_Goi")
      on SwitchOff: ResetBit("M_May_Dong_Goi")
      ProcessValue <- "M_May_Dong_Goi"
   Circle "Circle_1" at 169,654 size 76x76
      Appearance <- "Q_Lamp_Auto"
   Circle "Circle_2" at 302,654 size 76x76
      Appearance <- "Q_Lamp_Manu"
   Circle "Circle_3" at 435,654 size 76x76
      Appearance <- "Q_Lamp_Auto_Running"
   TextField "Text field_22" at 185,679 size 55x40; Text 'Auto'
   TextField "Text field_23" at 317,677 size 73x40; Text 'Manu'
   TextField "Text field_24" at 449,675 size 58x40; Text 'Run'
   Switch "Switch_4" at 318,295 size 89x40; TextOn 'ON'; CaptionText 'Switch'; TextOff 'OFF'; Authorization "khau1"
      on SwitchOff: ResetBit("M_Valve1")
      on SwitchOn: SetBit("M_Valve1")
      ProcessValue <- "M_Valve1"
   Button "Button_3" at 78,783 size 96x32; TextOff 'Screen1'
      on Click: ActivateScreen("Screen_1", 0)
   Button "Button_4" at 242,783 size 96x32; TextOff 'Screen2'
      on Click: ActivateScreen("Screen_2", 0)
   Switch "Switch_15" at 562,764 size 169x44; TextOn 'start'; CaptionText 'log data switches'; TextOff 'stop'
      on SwitchOff: function_b6526003(0, "Data_switches")
      on SwitchOn: function_fd9437ed(0, "Data_switches")
   Switch "Switch_16" at 784,764 size 169x44; TextOn 'start'; CaptionText 'log data temp'; TextOff 'stop'
      on SwitchOn: function_fd9437ed(0, "Data_temp")
      on SwitchOff: function_b6526003(0, "Data_temp")
   Button "Button_5" at 409,783 size 96x32; TextOff 'logout'
      on Click: function_f23ef4c9()

screen "Screen_2" 1440x900
   TextField "Text field_1" at 578,33 size 363x100; Text 'Screen phụ'
   AlarmView "Alarm view_1" at 170,122 size 1063x370
   Button "Button_1" at 465,560 size 186x128; TextOff 'alarm1'
      on Press: SetBit("alarm1")
      on Release: ResetBit("alarm1")
   Button "Button_2" at 762,560 size 186x128; TextOff 'alarm2'
      on Release: ResetBit("alarm2")
      on Press: SetBit("alarm2")
   Button "Button_3" at 495,728 size 96x32; TextOff 'Screen1'
      on Click: ActivateScreen("Screen_1", 0)
   Button "Button_4" at 659,728 size 96x32; TextOff 'Screen2'
      on Click: ActivateScreen("Screen_2", 0)
   Button "Button_5" at 828,728 size 96x32; TextOff 'logoff'
      on Click: function_f23ef4c9()
*)